// TwinCAT 3 PLC project Sample
// ProgramVersion: 3.1.4023.0
// libraries:
//   Tc2_Standard, * (Beckhoff Automation GmbH)
//   Tc2_System, * (Beckhoff Automation GmbH)
//   Tc3_Module, * (Beckhoff Automation GmbH)
// project tree:
//   / PlcTask.TcTTO
//   POUs/ MAIN.TcPOU
// real-time tasks:
//   TASK Device 1 (OPC UA Virtual)_Task_58: cycle T#40ms, priority 58, ADS port 350
//   TASK PlcTask: cycle T#10ms, priority 20, ADS port 351
// I/O:
//   DEVICE Device 1 (OPC UA Virtual), AmsNetId 192.168.56.1.2.1

CONFIGURATION Sample
    RESOURCE PLC ON TwinCAT3
        TASK PlcTask(INTERVAL := T#10ms, PRIORITY := 20);
        PROGRAM MAIN WITH PlcTask : MAIN;
    END_RESOURCE
END_CONFIGURATION

// ---- POUs/MAIN.TcPOU
PROGRAM MAIN
VAR
   fbWriteReq   : ADSWRITE := ( NETID := '127.0.0.1.1.1', PORT := 10, TMOUT := DEFAULT_ADS_TIMEOUT );
   bWrite       : BOOL; (* Rising edge at this variable starts command execution *)
   nState       : BYTE;
   bBusy        : BOOL;
   bError       : BOOL;
   nErrID       : UDINT;
   otcidOpcUaClient  : UDINT := 16#01010010;			(* TcCOM Objects -> Project Objects -> OTCID of respective IO Client Object *)
   ptcidServerUrl : UDINT := 16#03130002;				(* parameter value can be found in TMC -> 16#03130002 *)
   sEndpointUrl : STRING := 'opc.tcp://localhost:48030';(* New Server URL to be written to OPC UA I/O Client *)
   END_VAR

CASE nState OF
   0:
      IF bWrite THEN
         bWrite := FALSE;
         
         bBusy := TRUE;
         bError := FALSE;
         nErrID := 0;
         
         fbWriteReq( WRITE := FALSE );
         fbWriteReq( IDXGRP := otcidOpcUaClient, 
					 IDXOFFS := ptcidServerUrl, 
                  	 LEN := INT_TO_UDINT(LEN( sEndpointUrl )),
					 SRCADDR := ADR( sEndpointUrl ),
                  	 WRITE := TRUE );
					 
         nState := nState + 1;            
      END_IF
      
   1:
      fbWriteReq( WRITE := FALSE, BUSY=>bBusy, ERR=>bError, ERRID=>nErrID );
      IF NOT bBusy THEN
         IF NOT bError THEN
            nState := 0;(* Success *)
         ELSE
            nState := 100;(* Error *)
         END_IF
      END_IF

   100:(* TODO::Implement error handler *)
      nState := 0;
   
END_CASE

END_PROGRAM
